Fanuc KAREL source: VT_ACK_QUEUE.kl

PROGRAM T
%NOLOCKGROUP
VAR
 v0 : INTEGER
 v1 : INTEGER
 v2 : INTEGER
 v3 : INTEGER
BEGIN
 VT_ACK_QUEUE(v0, v1, v2, v3)
END T
